FUNCTION_BLOCK FB_realcontrolbox IMPLEMENTS I_controlbox
VAR_INPUT
END_VAR
VAR_OUTPUT
END_VAR
VAR
END_VAR

{warning 'add method implementation '}
METHOD Buttons
VAR_INPUT
	eModes	: E_Modes;
	eState	: E_States;
END_VAR
VAR_OUTPUT
	bStart	: BOOL;
	bStop	: BOOL;
END_VAR
END_METHOD

{warning 'add method implementation '}
METHOD Joystick
VAR_INPUT
	eModes	: E_Modes;
	eState	: E_Status;
END_VAR
VAR_OUTPUT
	fJoystickY	: LREAL;
	fJoystickX	: LREAL;
END_VAR
END_METHOD

{warning 'add method implementation '}
METHOD Lamps
VAR_INPUT
	eModes	: E_Modes;
	eState	: E_States;
END_VAR
END_METHOD

{warning 'add method implementation '}
METHOD Mode
VAR_OUTPUT
	eModes	: E_Modes;
END_VAR
END_METHOD

{warning 'add method implementation '}
METHOD State
VAR_INPUT
	eModes	: E_Modes;
END_VAR
VAR_OUTPUT
	eState	: E_States;
END_VAR
END_METHOD

END_FUNCTION_BLOCK

(* stored: Version 1.1.0.1, ProductVersion 3.1.4024.12
   POU FB_realcontrolbox: Id {684b9a4f-cee7-488b-a949-d1fe5216c95f}, SpecialFunc None
   Method Buttons: Id {13434b86-792c-487f-9b61-4ba600c4bae5}
   Method Joystick: Id {5301be79-c841-4db4-b709-15934a066227}
   Method Lamps: Id {b6637072-f1fd-496c-a4d6-c37fe870fa99}
   Method Mode: Id {3830b441-1d0b-457e-943a-fb56cee8a098}
   Method State: Id {87af71cf-e011-49dd-a643-c815f87dfadf} *)
